(* IEC 61131-3 sources: SmartHomeNew/SmartHomeNew-main/workspace/dut_rebuild/socket_v2/v2_core, 1 file *)

(* ---- FB_Socket_V2_Core_DRAFT.st ---- *)
FUNCTION_BLOCK FB_Socket_V2_Core_DRAFT
VAR_INPUT
    VI_Command : ST_Socket_Command_V2;
    VI_State_In : ST_Socket_State_V2;
END_VAR
VAR_OUTPUT
    VO_Command_Out : ST_Socket_Command_V2;
    VO_State_Out : ST_Socket_State_V2;
END_VAR

// Draft pass-through skeleton only.
VO_Command_Out := VI_Command;
VO_State_Out := VI_State_In;
END_FUNCTION_BLOCK
